// TIA Portal V14 export
FUNCTION "FC_DataProcess" : Void   // FC1, SCL
// stored: AutoNumber true
BEGIN
END_FUNCTION
